{attribute 'linkalways'} 
{attribute 'no_explicit_call' := 'This FB is a CLASS and must be accessed using methods or properties'}
{attribute 'enable_dynamic_creation'}
FUNCTION_BLOCK FINAL ADD_UINT EXTENDS Node
VAR
	in1 : _UINT(0);
	in2 : _UINT(0);
	out : _UINT(0);
END_VAR

METHOD PUBLIC Clone : I_Node
VAR
	pNode : POINTER TO ADD_UINT;
END_VAR
pNode := __NEW(ADD_UINT);
Clone := pNode^;
END_METHOD

METHOD FB_init : BOOL
VAR_INPUT
	bInitRetains : BOOL; // if TRUE, the retain variables are initialized (warm start / cold start)
	bInCopyCode : BOOL;  // if TRUE, the instance afterwards gets moved into the copy code (online change)
END_VAR
AddInput('in1',THIS^.in1);
AddInput('in2',THIS^.in2);
AddOutput('out', THIS^.out);
END_METHOD

METHOD PROTECTED OnExecute
VAR
END_VAR
out.Value := in1.Value + in2.Value;
END_METHOD

END_FUNCTION_BLOCK

(* stored: Version 1.1.0.1, ProductVersion 3.1.4024.15
   POU ADD_UINT: Id {9343a47a-fd9e-4d1d-8d1e-13c94d690c47}, SpecialFunc None
   Folder Constructor: Id {bbc1a2ab-f819-40c0-bdf5-59b16a1d350e}
   Method Clone: Id {a4ebb779-169b-4dc1-b64e-c910a2e13b88}
   Method FB_init: Id {6ab24b92-7e83-4485-8362-f315c7085a19}
   Method OnExecute: Id {76ce2dd5-1b6d-4b57-a478-c6f25e57f5e5} *)
